FUNCTION Set_Bit_F : BOOL
VAR_INPUT
	BIT_Number:  UINT;
END_VAR
VAR
END_VAR
VAR_IN_OUT
	Variavel: WORD;
END_VAR

// Set the bit
Variavel := Variavel OR SHL(WORD#1,BIT_Number);

END_FUNCTION

(* stored: Version 1.1.0.1
   POU Set_Bit_F: Id {aedeb09c-f1da-484a-814b-f14b895e9511}, SpecialFunc None *)
